TYPE TankCtrl_Io :
STRUCT
	in			: TankCtrl_Io_In;
	out			: TankCtrl_Io_Out;
END_STRUCT
END_TYPE

(* stored: Version 1.1.0.1
   DUT TankCtrl_Io: Id {3e2eae8d-e089-40d3-a315-94efb00e673c} *)
